// TwinCAT 3 PLC project Database_Library
// Title: Sqlite_Adaptor
// Company: Siang Poh
// ProjectVersion: 1.0
// ProgramVersion: 3.1.4020.10
// libraries:
//   Tc2_Database, * (Beckhoff Automation GmbH)
//   Tc2_Standard, * (Beckhoff Automation GmbH)
//   Tc2_System, * (Beckhoff Automation GmbH)
//   Tc3_Interfaces, * (Beckhoff Automation GmbH)
//   Tc3_Module, * (Beckhoff Automation GmbH)
// project tree:
//   Base Component/Class/ C_DBADAPTOR.TcPOU, C_SQLITECLIENT.TcPOU
//   Base Component/Custom Datatypes/ GVL_DATABASE_LIB.TcGVL, T_SQL_COMMAND.TcDUT
//   Base Component/Function/ GET_SQL_COMMAND_LENGTH.TcPOU
//   Version/ Global_Version.TcGVL
// (motion and I/O tree: see PLC project motion_library)
// real-time tasks:
//   TASK PlcTask: cycle T#10ms, priority 20, ADS port 350

// ---- Base Component/Custom Datatypes/T_SQL_COMMAND.TcDUT
TYPE T_SQL_COMMAND : STRING(GVL_DATABASE_LIB.MAX_SQL_LENGTH); END_TYPE

// ---- Base Component/Custom Datatypes/GVL_DATABASE_LIB.TcGVL
{attribute 'qualified_only'}
VAR_GLOBAL CONSTANT
	MAX_SQL_LENGTH : UDINT := 10000;
END_VAR

// ---- Version/Global_Version.TcGVL
// This function has been automatically generated from the project information.
VAR_GLOBAL CONSTANT
	{attribute 'const_non_replaced'}
	stLibVersion_Sqlite_Adaptor : ST_LibVersion := (iMajor := 1, iMinor := 0, iBuild := 0, iRevision := 0, sVersion := '1.0');
END_VAR

// ---- Base Component/Class/C_DBADAPTOR.TcPOU
//{attribute 'hide_all_locals'}
FUNCTION_BLOCK PUBLIC C_DBADAPTOR
VAR_INPUT
END_VAR
VAR_OUTPUT
END_VAR
VAR
	sAmsNetId	: STRING(23) := '';
	
	DB_ID		: UDINT := 0;
	isOpened	: BOOL := FALSE;
	
	_TIMEOUT	: TIME := T#3S;
	
	_FBOPENCONN	: FB_DBConnectionOpen;
	_FBCLOSECONN: FB_DBConnectionClose;
	_FBRELOAD	: FB_DBReloadConfig;
END_VAR

;

METHOD REACTIVATE_CONFIGURATION : DINT
VAR_INPUT
END_VAR
_FBRELOAD(
	sNetID:= sAmsNetID, 
	bExecute:= TRUE, 
	tTimeout:= _TIMEOUT, 
	bBusy=> , 
	bError=> , 
	nErrID=> );
IF _FBRELOAD.bError THEN
	_FBRELOAD(bExecute:= FALSE);
	REACTIVATE_CONFIGURATION := 1;
	RETURN;
ELSIF NOT _FBRELOAD.bBusy THEN
	_FBRELOAD(bExecute:= FALSE);
	REACTIVATE_CONFIGURATION := -1;
	RETURN;
ELSE
	REACTIVATE_CONFIGURATION := 0;
	RETURN;
END_IF
END_METHOD

{attribute 'object_name' := 'Close'}
METHOD CLOSE : DINT
VAR_INPUT
END_VAR
IF isOpened THEN
	_FBCLOSECONN(
		sNetID:= sAmsNetID, 
		hDBID:= DB_ID, 
		bExecute:= TRUE, 
		tTimeout:= _TIMEOUT );
	IF _FBCLOSECONN.bError THEN 
		_FBCLOSECONN(
			sNetID:= sAmsNetId, 
			hDBID:= DB_ID, 
			bExecute:= FALSE, 
			tTimeout:= _TIMEOUT );
		Close := 1;
		RETURN;
	ELSIF NOT _FBCLOSECONN.bBusy THEN
		_FBCLOSECONN(
			sNetID:= sAmsNetId, 
			hDBID:= DB_ID, 
			bExecute:= FALSE, 
			tTimeout:= _TIMEOUT );
		Close := -1;
		RETURN;
	ELSE
		Close := 0;
		RETURN;
	END_IF
ELSE
	CLOSE := 2;
	RETURN;
END_IF
END_METHOD

PROPERTY HANDLE : UDINT
SET
DB_ID := HANDLE;
END_SET
GET
HANDLE := DB_ID;
END_GET
END_PROPERTY

PROPERTY CONNECTION_OPENED : BOOL
GET
CONNECTION_OPENED := isOpened;
END_GET
END_PROPERTY

{attribute 'object_name' := 'Open'}
METHOD OPEN : DINT
VAR_INPUT
	DATABASE_HANDLE : UDINT;
END_VAR
IF NOT isOpened THEN
	_FBOPENCONN(
		sNetID:= sAmsNetId, 
		hDBID:= DATABASE_HANDLE, 
		bExecute:= TRUE, 
		tTimeout:= _TIMEOUT );
	IF _FBOPENCONN.bError THEN  
		_FBOPENCONN(
			sNetID:= sAmsNetId, 
			hDBID:= DB_ID, 
			bExecute:= FALSE, 
			tTimeout:= _TIMEOUT );
		OPEN := 1;
		RETURN;
	ELSIF NOT _FBOPENCONN.bBusy THEN
		_FBOPENCONN(
			sNetID:= sAmsNetId, 
			hDBID:= DB_ID, 
			bExecute:= FALSE, 
			tTimeout:= _TIMEOUT );
		isOpened := TRUE;
		DB_ID := DATABASE_HANDLE;
		Open := -1;
		RETURN;
	ELSE
		Open := 0;
		RETURN;
	END_IF
ELSE
	OPEN := 2;
	RETURN;
END_IF
END_METHOD

PROPERTY TIMEOUT : TIME
GET
TimeOut := _TIMEOUT;
END_GET
SET
_TIMEOUT := TimeOut;
END_SET
END_PROPERTY

END_FUNCTION_BLOCK

// ---- Base Component/Class/C_SQLITECLIENT.TcPOU
FUNCTION_BLOCK C_SQLITECLIENT EXTENDS C_DBADAPTOR
VAR_INPUT
END_VAR
VAR_OUTPUT
END_VAR
VAR
	_FBADDCONN		: FB_DBConnectionAdd;
	//_FBSQLDELETE 	: FB_DBRecordDelete;
	_FBSQLINSERT 	: FB_DBRecordInsert_EX;
	_FBSQLSELECT 	: FB_DBRecordArraySelect;
END_VAR

{attribute 'object_name' := 'SQL_EXECUTE_NONQUERY'}
METHOD SQL_EXECUTE_NONQUERY : DINT
VAR_INPUT
	SQL : POINTER TO T_SQL_COMMAND;
END_VAR
_FBSQLINSERT(
	sNetID:= sAmsNetId, 
	hDBID:= DB_ID, 
	pCmdAddr:= SQL, 
	cbCmdSize:= GET_SQL_COMMAND_LENGTH(SQL), 
	bExecute:= TRUE, 
	tTimeout:= _TIMEOUT );
IF _FBSQLINSERT.bError THEN
	_FBSQLINSERT(bExecute:= FALSE);
	SQL_EXECUTE_NONQUERY := 1;
	RETURN;
ELSIF NOT _FBSQLINSERT.bBusy THEN
	_FBSQLINSERT(bExecute:= FALSE);
	SQL_EXECUTE_NONQUERY := -1;
	RETURN;
ELSE
	SQL_EXECUTE_NONQUERY := 0;
	RETURN;
END_IF
END_METHOD

{attribute 'object_name' := 'SQL_EXECUTE_QUERY'}
METHOD SQL_EXECUTE_QUERY : DINT
VAR_INPUT
	SQL_PTR				: POINTER TO T_SQL_COMMAND;
	START_INDEX			: UDINT;
	ROWS_TO_READ		: UDINT;
	PTR_DATA_OUT		: PVOID;
	DATA_SIZE			: UDINT;
	DATABASE_ROWS		: POINTER TO UDINT;
END_VAR
_FBSQLSELECT(
	sNetID:= sAmsNetId, 
	hDBID:= DB_ID, 
	pCmdAddr:= SQL_PTR, 
	cbCmdSize:= GET_SQL_COMMAND_LENGTH(SQL_PTR), 
	nStartIndex:= START_INDEX, 
	nRecordCount:= ROWS_TO_READ, 
	pDestAddr:= PTR_DATA_OUT, 
	cbRecordArraySize:= DATA_SIZE, 
	bExecute:= TRUE, 
	tTimeout:= _TIMEOUT );
IF _FBSQLSELECT.bError THEN
	_FBSQLSELECT(bExecute:= FALSE);
	SQL_EXECUTE_QUERY := 1;
	RETURN;
ELSIF NOT _FBSQLSELECT.bBusy THEN
	DATABASE_ROWS^ := _FBSQLSELECT.nRecords;
	_FBSQLSELECT(bExecute:= FALSE);
	SQL_EXECUTE_QUERY := -1;
	RETURN;
ELSE 
	SQL_EXECUTE_QUERY := 0;
	RETURN;
END_IF
END_METHOD

METHOD CREATE_CONNECTION : DINT
VAR_INPUT
	URL					: STRING(255);
	TABLE				: STRING(255);
	NAME				: STRING(255);
	Database_Handle_Out : POINTER TO UDINT;	
END_VAR
_FBADDCONN(
	sNetID:= sAmsNetId, 
	eDBType:= eDBType_SQLite, 
	eDBValueType:= eDBValue_Bytes, 
	sDBServer:= NAME, 
	sDBUrl:= URL, 
	sDBTable:= TABLE, 
	bExecute:= TRUE, 
	tTimeout:= _TIMEOUT, 
	bBusy=> , 
	bError=> , 
	nErrID=> , 
	hDBID=> );
IF _FBADDCONN.bError THEN
	_FBADDCONN(bExecute:= FALSE);
	CREATE_CONNECTION := 1;
	RETURN; 
ELSIF NOT _FBADDCONN.bBusy THEN
	Database_Handle_Out^ := _FBADDCONN.hDBID;
	_FBADDCONN(bExecute:= FALSE);
	CREATE_CONNECTION := -1;
	RETURN; 
ELSE
	CREATE_CONNECTION := 0;
	RETURN;
END_IF
END_METHOD

END_FUNCTION_BLOCK

// ---- Base Component/Function/GET_SQL_COMMAND_LENGTH.TcPOU
FUNCTION GET_SQL_COMMAND_LENGTH : UDINT
VAR_INPUT
	COMMAND : POINTER TO T_SQL_COMMAND;
END_VAR
VAR
	_I 		: UDINT;
	_TEST 	: POINTER TO BYTE;
END_VAR

_TEST := COMMAND;
FOR _I := 0 TO (GVL_DATABASE_LIB.MAX_SQL_LENGTH) BY 1 DO
	IF _TEST[_I] = 0 THEN
		GET_SQL_COMMAND_LENGTH := _I;
		RETURN;
	END_IF
END_FOR

END_FUNCTION
